(* IEC 61131-3 sources: plc_simulator/services/codesys/GVLs, 4 files *)

(* ---- GVL_JC_Constants.st ---- *)
(* GVL_JC_Constants — Global constants *)
(* Identical names to globals.st VAR_GLOBAL CONSTANT — no renaming needed *)
VAR_GLOBAL CONSTANT

  (* ===== Layout Hierarchy Limits ===== *)
  MAX_LINES                 : INT  := 1;  (* max production lines in a plant *)
  MAX_STATIONS_PER_LINE     : INT  := 30;  (* max stations per line *)
  MAX_Transporters_PER_LINE : INT  := 3;  (* max transporters per line *)
  MIN_StationIndex          : INT  := 100;  (* first valid station index *)
  MAX_StationIndex          : INT  := 130;  (* MaxLines*100 + MaxStationsPerLine *)

  (* ===== Derived Absolute Limits ===== *)
  MAX_Transporters          : INT  := 3;  (* absolute max transporters in a plant *)
  MAX_Units                 : INT  := 10;  (* max units (lifting frames / hooks) *)
  MAX_STATIONS_PER_STEP     : INT  := 5;  (* max parallel stations per program stage *)
  MAX_STEPS_PER_PROGRAM     : INT  := 30;  (* max stages in a treatment program *)
  MAX_TASK_QUEUE            : INT  := 60;  (* max tasks per transporter queue *)

  (* ===== Algorithm / Scheduler Limits ===== *)
  DEP_MAX_IDLE_SLOTS        : INT  := 20;  (* max idle slots per transporter *)
  DEP_MAX_DELAY_ACTS        : INT  := 20;  (* max delay actions per cycle *)
  DEP_MAX_WAITING           : INT  := 5;  (* max waiting batches *)
  MIN_WorkingArea           : DINT := 20;  (* mm — TWA minimum working area *)

  (* ===== Scheduler Timing Constants ===== *)
  SCH_DISPATCH_MARGIN_S     : REAL := 3.0;  (* dispatch early-start margin (seconds) *)
  SCH_CONFLICT_MARGIN_S     : REAL := 1.0;  (* conflict detection margin (seconds) *)
  SCH_FLEX_FACTOR           : REAL := 0.5;  (* fraction of flex (max-cal) used by DEP *)
  SCH_MARGIN_S              : REAL := 5.0;  (* DEP small-delay threshold (seconds) *)
  SCH_MAX_INIT_WAIT_S       : REAL := 120.0;  (* max initial wait for stage0 pickup (seconds) *)
  SCH_END_DELAY_TICKS       : INT  := 100;  (* stabilization ticks after DEP activate *)
  SCH_MAX_FIT_ROUNDS        : INT  := 50;  (* max recalc rounds in DEP fit loop *)

  (* ===== Enumerated Constants ===== *)

  (* Unit status *)
  USED                      : INT  := 1;  (* unit in use *)
  NOT_USED                  : INT  := 0;  (* unit not in use *)

  (* Unit state *)
  EMPTY                     : INT  := 0;  (* unit is empty *)
  FULL                      : INT  := 1;  (* unit is full *)

  (* Unit target *)
  TO_NONE                   : INT  := 0;  (* no target *)
  TO_LOADING                : INT  := 1;  (* target: loading station *)
  TO_BUFFER                 : INT  := 2;  (* target: buffer station *)
  TO_PROCESS                : INT  := 3;  (* target: process station *)
  TO_UNLOAD                 : INT  := 4;  (* target: unloading station *)
  TO_AVOID                  : INT  := 5;  (* target: avoidance position *)

  (* Station kind *)
  KIND_DRY                  : INT  := 0;  (* dry station *)
  KIND_WET                  : INT  := 1;  (* wet station *)

  (* Station operation — logistics *)
  OP_BUFFER                 : INT  := 30;  (* buffer station *)
  OP_BUFFER_EMPTY           : INT  := 31;  (* empty buffer station *)
  OP_BUFFER_LOADED          : INT  := 32;  (* loaded buffer station *)
  OP_BUFFER_PROCESSED       : INT  := 33;  (* processed buffer station *)
  OP_LOADING                : INT  := 40;  (* loading operation *)
  OP_UNLOADING              : INT  := 41;  (* unloading operation *)
  OP_LOADING_UNLOADING      : INT  := 42;  (* combined loading/unloading *)

  (* Batch state *)
  NOT_PROCESSED             : INT  := 0;  (* batch not yet processed *)
  IN_PROCESS                : INT  := 1;  (* batch currently in process *)
  PROCESSED                 : INT  := 2;  (* batch processing complete *)

  (* Avoid status for stations (TWA) *)
  AVOID_None                : INT  := 0;  (* station not avoided *)
  AVOID_Passable            : INT  := 1;  (* pass through allowed, no stop *)
  AVOID_Block               : INT  := 2;  (* hard block, cannot pass *)

  (* Move-away constants *)
  MOVE_AWAY_MIN_WAIT_S      : LINT := 60;  (* don't start move-away if next task on same station starts within this many seconds *)
END_VAR

(* ---- GVL_JC_Parameters.st ---- *)
{attribute 'qualified_only'}
(* Scheduler GVL_Parameters — Production process data arrays *)
VAR_GLOBAL
  CountStations       : INT;                                                      (* configured station count *)
  Stations            : ARRAY[MIN_STATION_INDEX..MAX_STATION_INDEX] OF UDT_StationType;  (* station configuration *)
  StationOccupancy : ARRAY[1..MAX_STATION_INDEX] OF UDT_JC_UnitAtStationType;  (* unit location per station *)
  Transporters        : ARRAY[0..MAX_TRANSPORTERS] OF UDT_TransporterType;       (* transporter configuration, index 0 unused *)
  TransporterStatus       : ARRAY[1..MAX_TRANSPORTERS] OF UDT_TransporterStatusType; (* transporter runtime status *)
  Unit              : ARRAY[1..MAX_UNITS] OF UDT_JC_UnitType;                  (* unit (lifting frame) state *)
  Batch             : ARRAY[1..MAX_UNITS] OF UDT_BatchType;                    (* batch state per unit *)
  TreatmentPrograms   : ARRAY[1..MAX_UNITS] OF UDT_TreatmentProgramType;         (* treatment program per unit *)
  AvoidStatus      : ARRAY[MIN_STATION_INDEX..MAX_STATION_INDEX] OF INT;        (* AVOID_NONE/Passable/Block per station *)
END_VAR

(* ---- GVL_JC_Scheduler.st ---- *)
(* GVL_JC_Scheduler — Simulator-internal global variables *)
(* Identical names to globals.st VAR_GLOBAL — no renaming needed *)
VAR_GLOBAL
  (* ===== Simulation Transporter State ===== *)
  g_sim_trans                   : ARRAY[1..MAX_Transporters] OF UDT_JC_SimTransporterType;  (* physics + scheduler command state *)

  (* ===== No-Treatment Task Destinations ===== *)
  g_ntt                         : ARRAY[1..MAX_Transporters] OF UDT_JC_NttTransporterType;  (* no-treatment task destinations *)

  (* ===== Precomputed Movement Times ===== *)
  g_move                        : ARRAY[1..MAX_Transporters] OF UDT_JC_MoveTimesType;  (* precomputed movement times per transporter *)

  (* ===== Actual (Measured) Move Times ===== *)
  g_actual_move                 : ARRAY[1..MAX_Transporters] OF UDT_JC_ActualMoveTimeType;  (* phase timestamps updated after each completed task *)

  (* ===== Unit Schedule ===== *)
  g_schedule                    : ARRAY[1..MAX_Units] OF UDT_JC_TskScheduleType;  (* calculated schedule per unit *)

  (* ===== Task Queues ===== *)
  g_task                        : ARRAY[1..MAX_Transporters] OF UDT_JC_TskQueueType;  (* task queue per transporter *)

  (* ===== Departure Scheduler State ===== *)
  g_dep_wk_schedule             : ARRAY[1..MAX_Units] OF UDT_JC_TskScheduleType;  (* DEP workspace: schedules *)
  g_dep_wk_task                 : ARRAY[1..MAX_Transporters] OF UDT_JC_TskQueueType;  (* DEP workspace: task queues *)
  g_dep_wk_program              : ARRAY[1..MAX_Units] OF UDT_TreatmentProgramType;  (* DEP workspace: programs *)
  g_dep_wk_batch                : ARRAY[1..MAX_Units] OF UDT_BatchType;  (* DEP workspace: batch state *)
  g_dep_idle_slot               : ARRAY[1..MAX_Transporters] OF UDT_JC_DepIdleSlotSetType;  (* idle slots per transporter *)
  g_dep_waiting                 : ARRAY[1..DEP_MAX_WAITING] OF INT;  (* waiting batch unit indices *)
  g_dep_waiting_count           : INT;  (* number of waiting batches *)
  g_dep_overlap                 : UDT_JC_DepOverlapType;  (* overlap station flags *)
  g_dep_pending                 : UDT_JC_DepPendingWriteType;  (* ACTIVATE write buffer *)
  g_dep_activated               : BOOL;  (* handshake TSK ← DEP *)
  g_tsk_stable                  : BOOL;  (* tasksStableFlag: TRUE when last TSK cycle reached READY+conflict_free, cleared only on DEP activation/reset *)
  g_conflict_resolved           : BOOL;  (* TRUE when TSK Analyze found no conflicts — gate for DEP *)

  (* ===== Scheduler Debug Observability ===== *)
  g_sched_dbg_tsk_phase         : INT;  (* TSK scheduler current phase *)
  g_sched_dbg_dep_phase         : INT;  (* DEP scheduler current phase *)
  g_sched_dbg_turn              : INT;  (* 1=TSK ran, 2=DEP ran this cycle *)
  g_sched_dbg_skip_cnt          : INT;  (* DEP skip count *)
  g_sched_dbg_dep_reject_cnt    : INT;  (* DEP reject count this cycle *)
  g_sched_dbg_dep_fit_round     : INT;  (* DEP fit round counter *)
  g_sched_dbg_dep_cur_wait_unit : INT;  (* DEP current waiting batch unit *)
  g_sched_dbg_dep_wait_cnt      : INT;  (* DEP waiting batch count *)
  g_sched_dbg_batch_cnt         : INT;  (* TSK active batch count *)
  g_sched_dbg_tsk_round_ticks    : INT;  (* TSK ticks consumed by last completed round *)
  g_sched_dbg_dep_round_ticks    : INT;  (* DEP ticks consumed by last completed round *)

  (* ===== TSK Conflict Debug (non-LINT for OPC UA) ===== *)
  g_dbg_tsk_conflict_type       : INT;   (* last analyze: 0=none, 1=TASK_SEQ, 2=COLLISION, 3=HANDOFF *)
  g_dbg_tsk_conflict_iter       : INT;   (* resolve iterations this cycle *)
  g_dbg_tsk_conf_unit           : INT;   (* conflict task unit *)
  g_dbg_tsk_conf_stage          : INT;   (* conflict task stage *)
  g_dbg_tsk_blocked_unit        : INT;   (* blocked task unit *)
  g_dbg_tsk_blocked_stage       : INT;   (* blocked task stage *)
  g_dbg_tsk_deficit             : DINT;  (* last deficit in seconds *)
  g_dbg_tsk_stretch_cnt         : INT;   (* stretches applied this cycle *)
  g_dbg_tsk_total_adv           : DINT;  (* total advance seconds this cycle *)
  g_dbg_tsk_total_delay         : DINT;  (* total delay seconds this cycle *)
  g_dbg_prog_cal                : ARRAY[1..MAX_Units] OF DINT;  (* current stage CalTime snapshot per unit *)

  (* ===== Production Queue ===== *)
  g_production_queue            : INT;  (* 1=batches in queue, 0=queue empty *)

  (* ===== Unix Time ===== *)
  g_time_s                      : LINT;  (* absolute time in unix seconds *)
  g_time_100ms                  : LINT;  (* absolute time in 0.1s ticks *)
  g_time_sync                   : LINT;  (* gateway writes real unix seconds here at init *)
  g_time_offset                 : LINT;  (* g_time_sync - uptime_s at init *)

  (* ===== Event Queue ===== *)
  g_event                       : UDT_JC_EventQueueType;  (* circular event buffer *)
  g_event_pending               : UDT_JC_EventMsgType;  (* staging slot — written by other FBs *)
  g_event_pending_valid         : BOOL;  (* TRUE = pending message ready to enqueue *)
  g_event_ack_seq               : INT;   (* Gateway writes ack_seq via OPC UA to consume head message *)

  (* ===== UI Snapshot (SIM only — stable schedule for gateway reads) ===== *)
  g_sim_ui_schedule             : ARRAY[1..MAX_Units] OF UDT_JC_TskScheduleType;
  g_sim_ui_task                 : ARRAY[1..MAX_Transporters] OF UDT_JC_TskQueueType;
  g_sim_ui_wait_unit            : INT;   (* current waiting batch unit, 0 = none *)
  g_sim_ui_wait_reason          : INT;   (* 0=pending, 1=NO_SLOT, 2=DELAY_TOO_LARGE, 3=STATION_CONFLICT, 4=MAX_ROUNDS *)

  (* ===== Dispatched Task (Executor Input) ===== *)
  g_dispatched_task             : ARRAY[1..MAX_Transporters] OF UDT_JC_DispatchedTaskType;  (* filled by Dispatcher, read by Executor *)

  (* ===== Manual Task Commands ===== *)
  g_manual_task                 : ARRAY[1..MAX_Transporters] OF UDT_JC_ManualTaskType;  (* gateway writes, PLC clears Valid after execution *)

  (* ===== OPC UA Gateway Command Interface ===== *)
  (* Gateway writes g_cmd_code + g_cmd_param via OPC UA.
     PLC processes when g_cmd_code <> 0, then clears it.
     Commands:
       2 = init       (param = station_count)  — finalize config, start runtime
       3 = clear      — zero all config, stop runtime
  *)
  g_cmd_code                    : INT;   (* command code, non-zero = trigger *)
  g_cmd_param                   : INT;   (* command parameter *)
END_VAR

(* ---- GVL_Parameters.st ---- *)
(* GVL_Parameters — Production process data arrays *)
(* Identical names to globals.st VAR_GLOBAL — no renaming needed *)
VAR_GLOBAL
  CountStations                  : INT;  (* configured station count *)
  Stations                     : ARRAY[MIN_StationIndex..MAX_StationIndex] OF UDT_StationType;  (* station configuration *)
  g_station_loc                 : ARRAY[1..MAX_StationIndex] OF UDT_UnitLocation;  (* unit location per station *)
  Transporters                         : ARRAY[0..MAX_Transporters] OF UDT_TransporterType;  (* transporter configuration, index 0 unused *)
  g_transporter                 : ARRAY[1..MAX_Transporters] OF UDT_TransporterStatusType;  (* transporter runtime status *)
  g_unit                        : ARRAY[1..MAX_Units] OF UDT_UnitType;  (* unit (lifting frame) state *)
  g_batch                       : ARRAY[1..MAX_Units] OF UDT_BatchType;  (* batch state per unit *)
  TreatmentPrograms                     : ARRAY[1..MAX_Units] OF UDT_TreatmentProgramType;  (* treatment program per unit *)
  g_avoid_status                : ARRAY[MIN_StationIndex..MAX_StationIndex] OF INT;  (* AVOID_None/Passable/Block per station *)
END_VAR
